REGION Network 21: UNIT 02 FIXTURE 2 PART A PRESENT
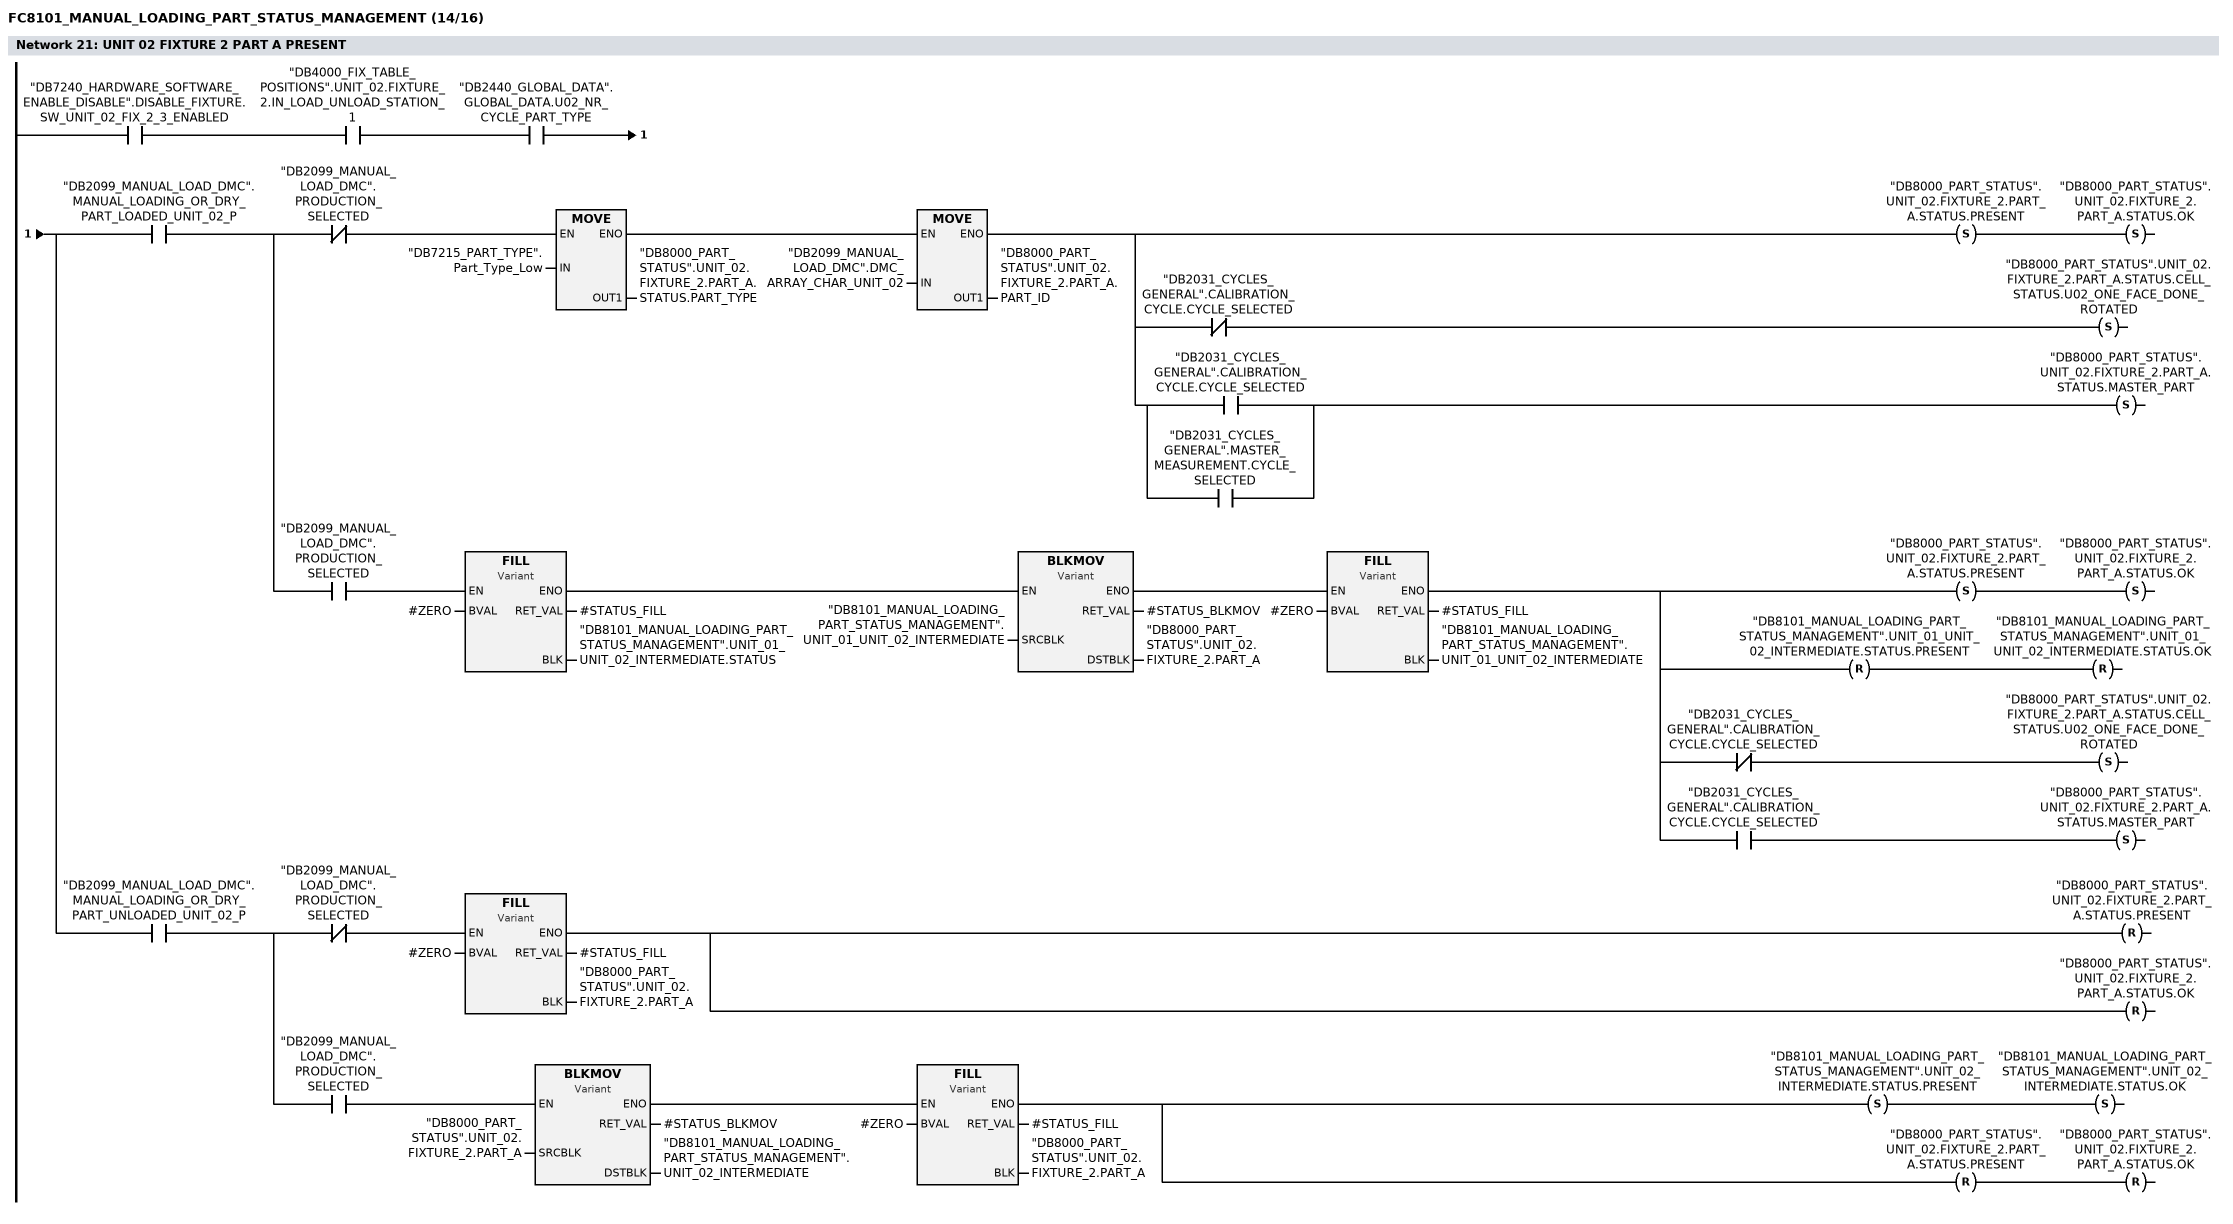
   RUNG wire#powerrail
      Contact( "DB7240_HARDWARE_SOFTWARE_ENABLE_DISABLE".DISABLE_FIXTURE.SW_UNIT_02_FIX_2_3_ENABLED )
      Contact( "DB4000_FIX_TABLE_POSITIONS".UNIT_02.FIXTURE_2.IN_LOAD_UNLOAD_STATION_1 )
      Contact( "DB2440_GLOBAL_DATA".GLOBAL_DATA.U02_NR_CYCLE_PART_TYPE )
      wire#w1
      Contact( "DB2099_MANUAL_LOAD_DMC".MANUAL_LOADING_OR_DRY_PART_LOADED_UNIT_02_P )
      wire#w2
      I_Contact( "DB2099_MANUAL_LOAD_DMC".PRODUCTION_SELECTED )
      { S7_GenerateENO := "TRUE" } Move(in := "DB7215_PART_TYPE".Part_Type_Low, out1 => "DB8000_PART_STATUS".UNIT_02.FIXTURE_2.PART_A.STATUS.PART_TYPE)
      Move(in := "DB2099_MANUAL_LOAD_DMC".DMC_ARRAY_CHAR_UNIT_02, out1 => "DB8000_PART_STATUS".UNIT_02.FIXTURE_2.PART_A.PART_ID)
      wire#w3
      S_Coil( "DB8000_PART_STATUS".UNIT_02.FIXTURE_2.PART_A.STATUS.PRESENT )
      S_Coil( "DB8000_PART_STATUS".UNIT_02.FIXTURE_2.PART_A.STATUS.OK )
   END_RUNG
   RUNG wire#w3
      I_Contact( "DB2031_CYCLES_GENERAL".CALIBRATION_CYCLE.CYCLE_SELECTED )
      S_Coil( "DB8000_PART_STATUS".UNIT_02.FIXTURE_2.PART_A.STATUS.CELL_STATUS.U02_ONE_FACE_DONE_ROTATED )
   END_RUNG
   RUNG wire#w3
      Contact( "DB2031_CYCLES_GENERAL".CALIBRATION_CYCLE.CYCLE_SELECTED )
      wire#w4
      S_Coil( "DB8000_PART_STATUS".UNIT_02.FIXTURE_2.PART_A.STATUS.MASTER_PART )
   END_RUNG
   RUNG wire#w3
      Contact( "DB2031_CYCLES_GENERAL".MASTER_MEASUREMENT.CYCLE_SELECTED )
   END_RUNG wire#w4
   RUNG wire#w2
      Contact( "DB2099_MANUAL_LOAD_DMC".PRODUCTION_SELECTED )
      { S7_Templates := "ptr_type := Variant" } FILL(BVAL := #ZERO, RET_VAL => #STATUS_FILL, BLK => "DB8101_MANUAL_LOADING_PART_STATUS_MANAGEMENT".UNIT_01_UNIT_02_INTERMEDIATE.STATUS)
      { S7_Templates := "blk_type := Variant" } BLKMOV(SRCBLK := "DB8101_MANUAL_LOADING_PART_STATUS_MANAGEMENT".UNIT_01_UNIT_02_INTERMEDIATE, RET_VAL => #STATUS_BLKMOV, DSTBLK => "DB8000_PART_STATUS".UNIT_02.FIXTURE_2.PART_A)
      { S7_Templates := "ptr_type := Variant" } FILL(BVAL := #ZERO, RET_VAL => #STATUS_FILL, BLK => "DB8101_MANUAL_LOADING_PART_STATUS_MANAGEMENT".UNIT_01_UNIT_02_INTERMEDIATE)
      wire#w5
      S_Coil( "DB8000_PART_STATUS".UNIT_02.FIXTURE_2.PART_A.STATUS.PRESENT )
      S_Coil( "DB8000_PART_STATUS".UNIT_02.FIXTURE_2.PART_A.STATUS.OK )
   END_RUNG
   RUNG wire#w5
      R_Coil( "DB8101_MANUAL_LOADING_PART_STATUS_MANAGEMENT".UNIT_01_UNIT_02_INTERMEDIATE.STATUS.PRESENT )
      R_Coil( "DB8101_MANUAL_LOADING_PART_STATUS_MANAGEMENT".UNIT_01_UNIT_02_INTERMEDIATE.STATUS.OK )
   END_RUNG
   RUNG wire#w5
      I_Contact( "DB2031_CYCLES_GENERAL".CALIBRATION_CYCLE.CYCLE_SELECTED )
      S_Coil( "DB8000_PART_STATUS".UNIT_02.FIXTURE_2.PART_A.STATUS.CELL_STATUS.U02_ONE_FACE_DONE_ROTATED )
   END_RUNG
   RUNG wire#w5
      Contact( "DB2031_CYCLES_GENERAL".CALIBRATION_CYCLE.CYCLE_SELECTED )
      S_Coil( "DB8000_PART_STATUS".UNIT_02.FIXTURE_2.PART_A.STATUS.MASTER_PART )
   END_RUNG
   RUNG wire#w1
      Contact( "DB2099_MANUAL_LOAD_DMC".MANUAL_LOADING_OR_DRY_PART_UNLOADED_UNIT_02_P )
      wire#w6
      I_Contact( "DB2099_MANUAL_LOAD_DMC".PRODUCTION_SELECTED )
      { S7_Templates := "ptr_type := Variant" } FILL(BVAL := #ZERO, RET_VAL => #STATUS_FILL, BLK => "DB8000_PART_STATUS".UNIT_02.FIXTURE_2.PART_A)
      wire#w7
      R_Coil( "DB8000_PART_STATUS".UNIT_02.FIXTURE_2.PART_A.STATUS.PRESENT )
   END_RUNG
   RUNG wire#w7
      R_Coil( "DB8000_PART_STATUS".UNIT_02.FIXTURE_2.PART_A.STATUS.OK )
   END_RUNG
   RUNG wire#w6
      Contact( "DB2099_MANUAL_LOAD_DMC".PRODUCTION_SELECTED )
      { S7_Templates := "blk_type := Variant" } BLKMOV(SRCBLK := "DB8000_PART_STATUS".UNIT_02.FIXTURE_2.PART_A, RET_VAL => #STATUS_BLKMOV, DSTBLK => "DB8101_MANUAL_LOADING_PART_STATUS_MANAGEMENT".UNIT_02_INTERMEDIATE)
      { S7_Templates := "ptr_type := Variant" } FILL(BVAL := #ZERO, RET_VAL => #STATUS_FILL, BLK => "DB8000_PART_STATUS".UNIT_02.FIXTURE_2.PART_A)
      wire#w8
      S_Coil( "DB8101_MANUAL_LOADING_PART_STATUS_MANAGEMENT".UNIT_02_INTERMEDIATE.STATUS.PRESENT )
      S_Coil( "DB8101_MANUAL_LOADING_PART_STATUS_MANAGEMENT".UNIT_02_INTERMEDIATE.STATUS.OK )
   END_RUNG
   RUNG wire#w8
      R_Coil( "DB8000_PART_STATUS".UNIT_02.FIXTURE_2.PART_A.STATUS.PRESENT )
      R_Coil( "DB8000_PART_STATUS".UNIT_02.FIXTURE_2.PART_A.STATUS.OK )
   END_RUNG
   // the same network as SCL:
   // ENO of a box is taken as its EN; it also drops when the box reports an error
   #_w1 := "DB7240_HARDWARE_SOFTWARE_ENABLE_DISABLE".DISABLE_FIXTURE.SW_UNIT_02_FIX_2_3_ENABLED AND "DB4000_FIX_TABLE_POSITIONS".UNIT_02.FIXTURE_2.IN_LOAD_UNLOAD_STATION_1 AND "DB2440_GLOBAL_DATA".GLOBAL_DATA.U02_NR_CYCLE_PART_TYPE;
   #_w2 := #_w1 AND "DB2099_MANUAL_LOAD_DMC".MANUAL_LOADING_OR_DRY_PART_LOADED_UNIT_02_P;
   #_w3 := #_w2 AND NOT "DB2099_MANUAL_LOAD_DMC".PRODUCTION_SELECTED;
   IF #_w3 THEN
       "DB8000_PART_STATUS".UNIT_02.FIXTURE_2.PART_A.STATUS.PART_TYPE := "DB7215_PART_TYPE".Part_Type_Low;
       "DB8000_PART_STATUS".UNIT_02.FIXTURE_2.PART_A.PART_ID := "DB2099_MANUAL_LOAD_DMC".DMC_ARRAY_CHAR_UNIT_02;
       "DB8000_PART_STATUS".UNIT_02.FIXTURE_2.PART_A.STATUS.PRESENT := TRUE;
       "DB8000_PART_STATUS".UNIT_02.FIXTURE_2.PART_A.STATUS.OK := TRUE;
   END_IF;
   IF #_w3 AND NOT "DB2031_CYCLES_GENERAL".CALIBRATION_CYCLE.CYCLE_SELECTED THEN
       "DB8000_PART_STATUS".UNIT_02.FIXTURE_2.PART_A.STATUS.CELL_STATUS.U02_ONE_FACE_DONE_ROTATED := TRUE;
   END_IF;
   IF #_w3 AND ("DB2031_CYCLES_GENERAL".CALIBRATION_CYCLE.CYCLE_SELECTED OR "DB2031_CYCLES_GENERAL".MASTER_MEASUREMENT.CYCLE_SELECTED) THEN
       "DB8000_PART_STATUS".UNIT_02.FIXTURE_2.PART_A.STATUS.MASTER_PART := TRUE;
   END_IF;
   #_w4 := #_w2 AND "DB2099_MANUAL_LOAD_DMC".PRODUCTION_SELECTED;
   #STATUS_FILL := FILL(EN := #_w4,
                        BVAL := #ZERO,
                        BLK => "DB8101_MANUAL_LOADING_PART_STATUS_MANAGEMENT".UNIT_01_UNIT_02_INTERMEDIATE.STATUS,
                        ENO => #_w5);
   #STATUS_BLKMOV := BLKMOV(EN := #_w5,
                           SRCBLK := "DB8101_MANUAL_LOADING_PART_STATUS_MANAGEMENT".UNIT_01_UNIT_02_INTERMEDIATE,
                           DSTBLK => "DB8000_PART_STATUS".UNIT_02.FIXTURE_2.PART_A,
                           ENO => #_w6);
   #STATUS_FILL := FILL(EN := #_w6,
                        BVAL := #ZERO,
                        BLK => "DB8101_MANUAL_LOADING_PART_STATUS_MANAGEMENT".UNIT_01_UNIT_02_INTERMEDIATE,
                        ENO => #_w7);
   IF #_w7 THEN
       "DB8000_PART_STATUS".UNIT_02.FIXTURE_2.PART_A.STATUS.PRESENT := TRUE;
       "DB8000_PART_STATUS".UNIT_02.FIXTURE_2.PART_A.STATUS.OK := TRUE;
       "DB8101_MANUAL_LOADING_PART_STATUS_MANAGEMENT".UNIT_01_UNIT_02_INTERMEDIATE.STATUS.PRESENT := FALSE;
       "DB8101_MANUAL_LOADING_PART_STATUS_MANAGEMENT".UNIT_01_UNIT_02_INTERMEDIATE.STATUS.OK := FALSE;
   END_IF;
   IF #_w7 AND NOT "DB2031_CYCLES_GENERAL".CALIBRATION_CYCLE.CYCLE_SELECTED THEN
       "DB8000_PART_STATUS".UNIT_02.FIXTURE_2.PART_A.STATUS.CELL_STATUS.U02_ONE_FACE_DONE_ROTATED := TRUE;
   END_IF;
   IF #_w7 AND "DB2031_CYCLES_GENERAL".CALIBRATION_CYCLE.CYCLE_SELECTED THEN
       "DB8000_PART_STATUS".UNIT_02.FIXTURE_2.PART_A.STATUS.MASTER_PART := TRUE;
   END_IF;
   #_w8 := #_w1 AND "DB2099_MANUAL_LOAD_DMC".MANUAL_LOADING_OR_DRY_PART_UNLOADED_UNIT_02_P;
   #STATUS_FILL := FILL(EN := #_w8 AND NOT "DB2099_MANUAL_LOAD_DMC".PRODUCTION_SELECTED,
                        BVAL := #ZERO,
                        BLK => "DB8000_PART_STATUS".UNIT_02.FIXTURE_2.PART_A,
                        ENO => #_w9);
   IF #_w9 THEN
       "DB8000_PART_STATUS".UNIT_02.FIXTURE_2.PART_A.STATUS.PRESENT := FALSE;
       "DB8000_PART_STATUS".UNIT_02.FIXTURE_2.PART_A.STATUS.OK := FALSE;
   END_IF;
   #STATUS_BLKMOV := BLKMOV(EN := #_w8 AND "DB2099_MANUAL_LOAD_DMC".PRODUCTION_SELECTED,
                           SRCBLK := "DB8000_PART_STATUS".UNIT_02.FIXTURE_2.PART_A,
                           DSTBLK => "DB8101_MANUAL_LOADING_PART_STATUS_MANAGEMENT".UNIT_02_INTERMEDIATE,
                           ENO => #_w10);
   #STATUS_FILL := FILL(EN := #_w10,
                        BVAL := #ZERO,
                        BLK => "DB8000_PART_STATUS".UNIT_02.FIXTURE_2.PART_A,
                        ENO => #_w11);
   IF #_w11 THEN
       "DB8101_MANUAL_LOADING_PART_STATUS_MANAGEMENT".UNIT_02_INTERMEDIATE.STATUS.PRESENT := TRUE;
       "DB8101_MANUAL_LOADING_PART_STATUS_MANAGEMENT".UNIT_02_INTERMEDIATE.STATUS.OK := TRUE;
       "DB8000_PART_STATUS".UNIT_02.FIXTURE_2.PART_A.STATUS.PRESENT := FALSE;
       "DB8000_PART_STATUS".UNIT_02.FIXTURE_2.PART_A.STATUS.OK := FALSE;
   END_IF;
END_REGION

REGION Network 22: UNIT 02 FIXTURE 3 PART A PRESENT
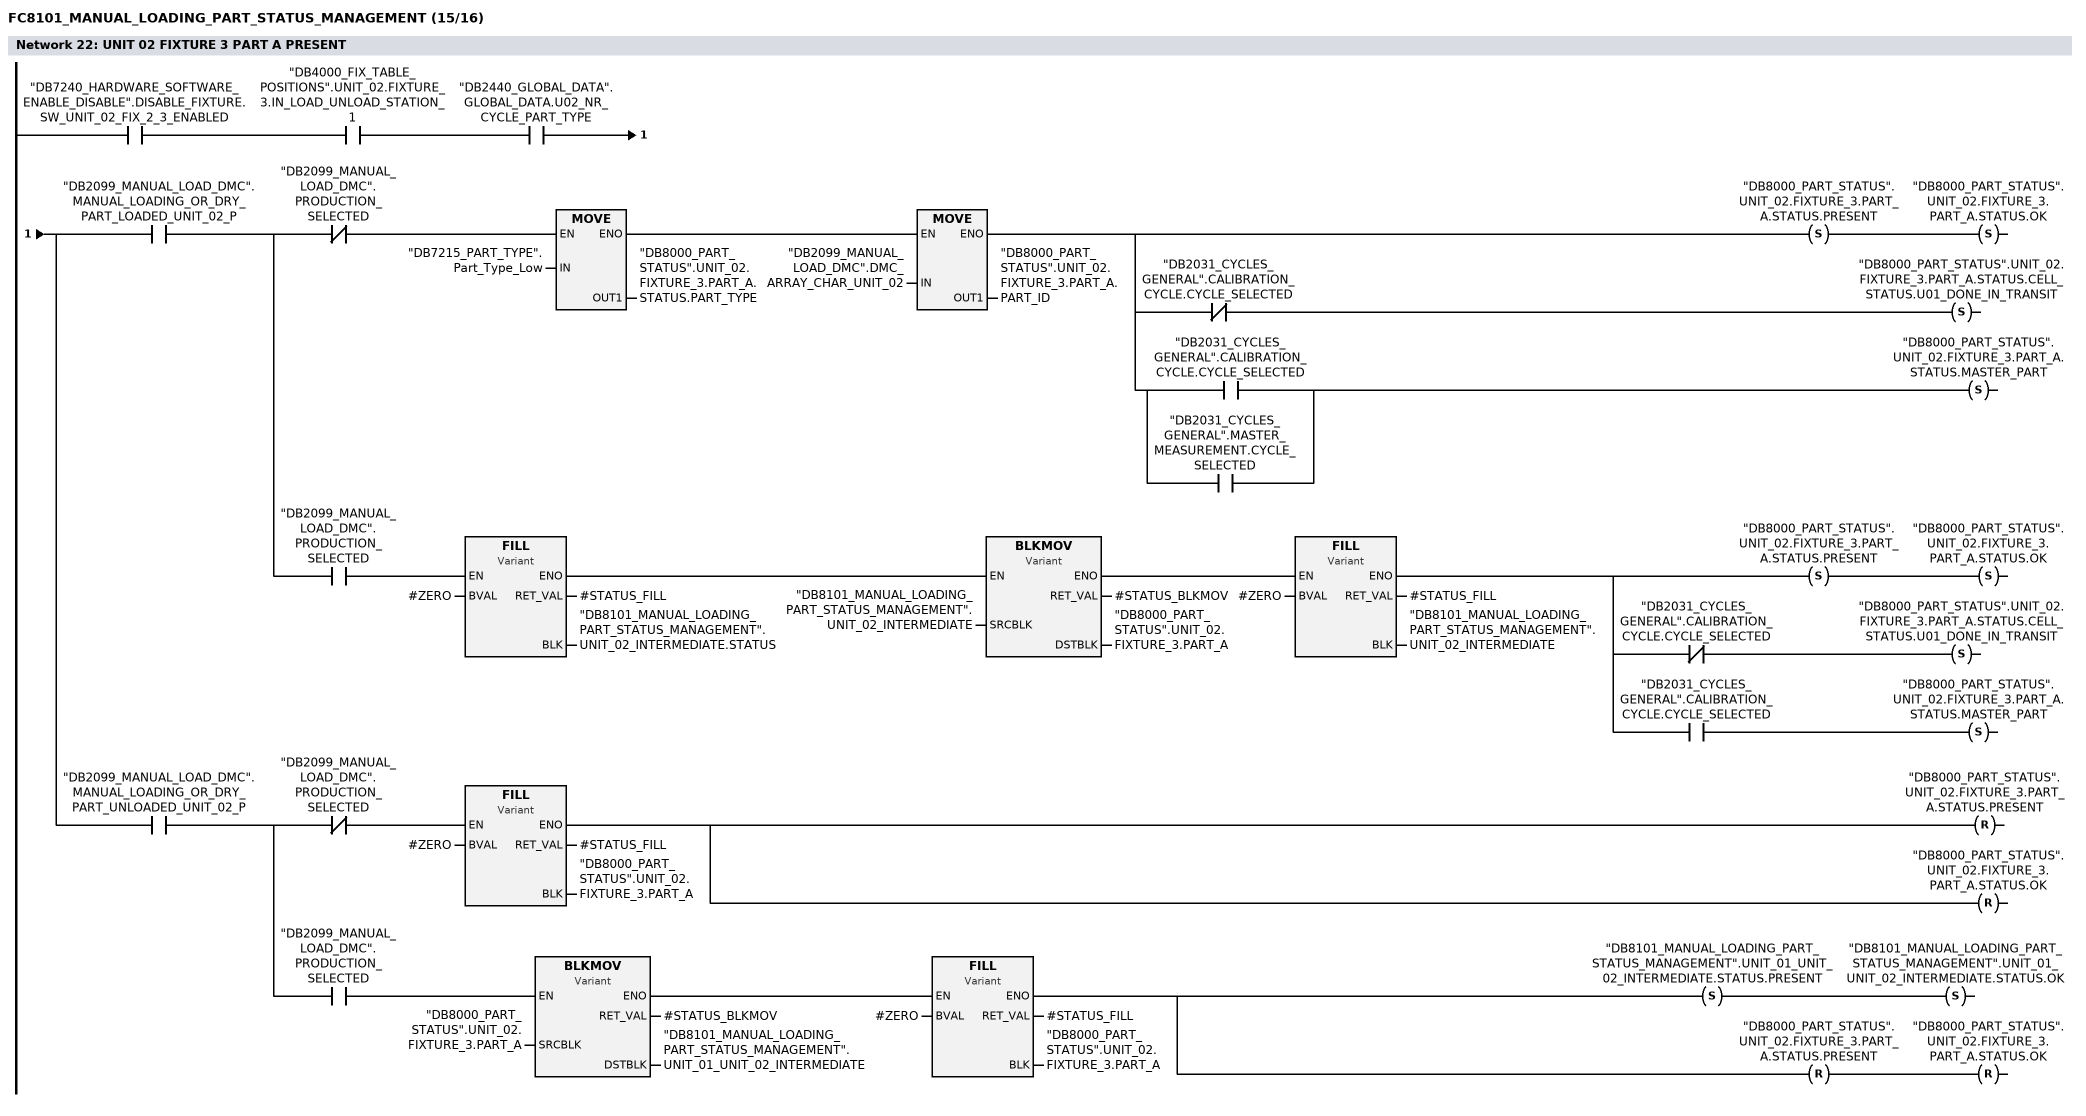
   RUNG wire#powerrail
      Contact( "DB7240_HARDWARE_SOFTWARE_ENABLE_DISABLE".DISABLE_FIXTURE.SW_UNIT_02_FIX_2_3_ENABLED )
      Contact( "DB4000_FIX_TABLE_POSITIONS".UNIT_02.FIXTURE_3.IN_LOAD_UNLOAD_STATION_1 )
      Contact( "DB2440_GLOBAL_DATA".GLOBAL_DATA.U02_NR_CYCLE_PART_TYPE )
      wire#w1
      Contact( "DB2099_MANUAL_LOAD_DMC".MANUAL_LOADING_OR_DRY_PART_LOADED_UNIT_02_P )
      wire#w2
      I_Contact( "DB2099_MANUAL_LOAD_DMC".PRODUCTION_SELECTED )
      { S7_GenerateENO := "TRUE" } Move(in := "DB7215_PART_TYPE".Part_Type_Low, out1 => "DB8000_PART_STATUS".UNIT_02.FIXTURE_3.PART_A.STATUS.PART_TYPE)
      Move(in := "DB2099_MANUAL_LOAD_DMC".DMC_ARRAY_CHAR_UNIT_02, out1 => "DB8000_PART_STATUS".UNIT_02.FIXTURE_3.PART_A.PART_ID)
      wire#w3
      S_Coil( "DB8000_PART_STATUS".UNIT_02.FIXTURE_3.PART_A.STATUS.PRESENT )
      S_Coil( "DB8000_PART_STATUS".UNIT_02.FIXTURE_3.PART_A.STATUS.OK )
   END_RUNG
   RUNG wire#w3
      I_Contact( "DB2031_CYCLES_GENERAL".CALIBRATION_CYCLE.CYCLE_SELECTED )
      S_Coil( "DB8000_PART_STATUS".UNIT_02.FIXTURE_3.PART_A.STATUS.CELL_STATUS.U01_DONE_IN_TRANSIT )
   END_RUNG
   RUNG wire#w3
      Contact( "DB2031_CYCLES_GENERAL".CALIBRATION_CYCLE.CYCLE_SELECTED )
      wire#w4
      S_Coil( "DB8000_PART_STATUS".UNIT_02.FIXTURE_3.PART_A.STATUS.MASTER_PART )
   END_RUNG
   RUNG wire#w3
      Contact( "DB2031_CYCLES_GENERAL".MASTER_MEASUREMENT.CYCLE_SELECTED )
   END_RUNG wire#w4
   RUNG wire#w2
      Contact( "DB2099_MANUAL_LOAD_DMC".PRODUCTION_SELECTED )
      { S7_Templates := "ptr_type := Variant" } FILL(BVAL := #ZERO, RET_VAL => #STATUS_FILL, BLK => "DB8101_MANUAL_LOADING_PART_STATUS_MANAGEMENT".UNIT_02_INTERMEDIATE.STATUS)
      { S7_Templates := "blk_type := Variant" } BLKMOV(SRCBLK := "DB8101_MANUAL_LOADING_PART_STATUS_MANAGEMENT".UNIT_02_INTERMEDIATE, RET_VAL => #STATUS_BLKMOV, DSTBLK => "DB8000_PART_STATUS".UNIT_02.FIXTURE_3.PART_A)
      { S7_Templates := "ptr_type := Variant" } FILL(BVAL := #ZERO, RET_VAL => #STATUS_FILL, BLK => "DB8101_MANUAL_LOADING_PART_STATUS_MANAGEMENT".UNIT_02_INTERMEDIATE)
      wire#w5
      S_Coil( "DB8000_PART_STATUS".UNIT_02.FIXTURE_3.PART_A.STATUS.PRESENT )
      S_Coil( "DB8000_PART_STATUS".UNIT_02.FIXTURE_3.PART_A.STATUS.OK )
   END_RUNG
   RUNG wire#w5
      I_Contact( "DB2031_CYCLES_GENERAL".CALIBRATION_CYCLE.CYCLE_SELECTED )
      S_Coil( "DB8000_PART_STATUS".UNIT_02.FIXTURE_3.PART_A.STATUS.CELL_STATUS.U01_DONE_IN_TRANSIT )
   END_RUNG
   RUNG wire#w5
      Contact( "DB2031_CYCLES_GENERAL".CALIBRATION_CYCLE.CYCLE_SELECTED )
      S_Coil( "DB8000_PART_STATUS".UNIT_02.FIXTURE_3.PART_A.STATUS.MASTER_PART )
   END_RUNG
   RUNG wire#w1
      Contact( "DB2099_MANUAL_LOAD_DMC".MANUAL_LOADING_OR_DRY_PART_UNLOADED_UNIT_02_P )
      wire#w6
      I_Contact( "DB2099_MANUAL_LOAD_DMC".PRODUCTION_SELECTED )
      { S7_Templates := "ptr_type := Variant" } FILL(BVAL := #ZERO, RET_VAL => #STATUS_FILL, BLK => "DB8000_PART_STATUS".UNIT_02.FIXTURE_3.PART_A)
      wire#w7
      R_Coil( "DB8000_PART_STATUS".UNIT_02.FIXTURE_3.PART_A.STATUS.PRESENT )
   END_RUNG
   RUNG wire#w7
      R_Coil( "DB8000_PART_STATUS".UNIT_02.FIXTURE_3.PART_A.STATUS.OK )
   END_RUNG
   RUNG wire#w6
      Contact( "DB2099_MANUAL_LOAD_DMC".PRODUCTION_SELECTED )
      { S7_Templates := "blk_type := Variant" } BLKMOV(SRCBLK := "DB8000_PART_STATUS".UNIT_02.FIXTURE_3.PART_A, RET_VAL => #STATUS_BLKMOV, DSTBLK => "DB8101_MANUAL_LOADING_PART_STATUS_MANAGEMENT".UNIT_01_UNIT_02_INTERMEDIATE)
      { S7_Templates := "ptr_type := Variant" } FILL(BVAL := #ZERO, RET_VAL => #STATUS_FILL, BLK => "DB8000_PART_STATUS".UNIT_02.FIXTURE_3.PART_A)
      wire#w8
      S_Coil( "DB8101_MANUAL_LOADING_PART_STATUS_MANAGEMENT".UNIT_01_UNIT_02_INTERMEDIATE.STATUS.PRESENT )
      S_Coil( "DB8101_MANUAL_LOADING_PART_STATUS_MANAGEMENT".UNIT_01_UNIT_02_INTERMEDIATE.STATUS.OK )
   END_RUNG
   RUNG wire#w8
      R_Coil( "DB8000_PART_STATUS".UNIT_02.FIXTURE_3.PART_A.STATUS.PRESENT )
      R_Coil( "DB8000_PART_STATUS".UNIT_02.FIXTURE_3.PART_A.STATUS.OK )
   END_RUNG
   // the same network as SCL:
   // ENO of a box is taken as its EN; it also drops when the box reports an error
   #_w1 := "DB7240_HARDWARE_SOFTWARE_ENABLE_DISABLE".DISABLE_FIXTURE.SW_UNIT_02_FIX_2_3_ENABLED AND "DB4000_FIX_TABLE_POSITIONS".UNIT_02.FIXTURE_3.IN_LOAD_UNLOAD_STATION_1 AND "DB2440_GLOBAL_DATA".GLOBAL_DATA.U02_NR_CYCLE_PART_TYPE;
   #_w2 := #_w1 AND "DB2099_MANUAL_LOAD_DMC".MANUAL_LOADING_OR_DRY_PART_LOADED_UNIT_02_P;
   #_w3 := #_w2 AND NOT "DB2099_MANUAL_LOAD_DMC".PRODUCTION_SELECTED;
   IF #_w3 THEN
       "DB8000_PART_STATUS".UNIT_02.FIXTURE_3.PART_A.STATUS.PART_TYPE := "DB7215_PART_TYPE".Part_Type_Low;
       "DB8000_PART_STATUS".UNIT_02.FIXTURE_3.PART_A.PART_ID := "DB2099_MANUAL_LOAD_DMC".DMC_ARRAY_CHAR_UNIT_02;
       "DB8000_PART_STATUS".UNIT_02.FIXTURE_3.PART_A.STATUS.PRESENT := TRUE;
       "DB8000_PART_STATUS".UNIT_02.FIXTURE_3.PART_A.STATUS.OK := TRUE;
   END_IF;
   IF #_w3 AND NOT "DB2031_CYCLES_GENERAL".CALIBRATION_CYCLE.CYCLE_SELECTED THEN
       "DB8000_PART_STATUS".UNIT_02.FIXTURE_3.PART_A.STATUS.CELL_STATUS.U01_DONE_IN_TRANSIT := TRUE;
   END_IF;
   IF #_w3 AND ("DB2031_CYCLES_GENERAL".CALIBRATION_CYCLE.CYCLE_SELECTED OR "DB2031_CYCLES_GENERAL".MASTER_MEASUREMENT.CYCLE_SELECTED) THEN
       "DB8000_PART_STATUS".UNIT_02.FIXTURE_3.PART_A.STATUS.MASTER_PART := TRUE;
   END_IF;
   #_w4 := #_w2 AND "DB2099_MANUAL_LOAD_DMC".PRODUCTION_SELECTED;
   #STATUS_FILL := FILL(EN := #_w4,
                        BVAL := #ZERO,
                        BLK => "DB8101_MANUAL_LOADING_PART_STATUS_MANAGEMENT".UNIT_02_INTERMEDIATE.STATUS,
                        ENO => #_w5);
   #STATUS_BLKMOV := BLKMOV(EN := #_w5,
                           SRCBLK := "DB8101_MANUAL_LOADING_PART_STATUS_MANAGEMENT".UNIT_02_INTERMEDIATE,
                           DSTBLK => "DB8000_PART_STATUS".UNIT_02.FIXTURE_3.PART_A,
                           ENO => #_w6);
   #STATUS_FILL := FILL(EN := #_w6,
                        BVAL := #ZERO,
                        BLK => "DB8101_MANUAL_LOADING_PART_STATUS_MANAGEMENT".UNIT_02_INTERMEDIATE,
                        ENO => #_w7);
   IF #_w7 THEN
       "DB8000_PART_STATUS".UNIT_02.FIXTURE_3.PART_A.STATUS.PRESENT := TRUE;
       "DB8000_PART_STATUS".UNIT_02.FIXTURE_3.PART_A.STATUS.OK := TRUE;
   END_IF;
   IF #_w7 AND NOT "DB2031_CYCLES_GENERAL".CALIBRATION_CYCLE.CYCLE_SELECTED THEN
       "DB8000_PART_STATUS".UNIT_02.FIXTURE_3.PART_A.STATUS.CELL_STATUS.U01_DONE_IN_TRANSIT := TRUE;
   END_IF;
   IF #_w7 AND "DB2031_CYCLES_GENERAL".CALIBRATION_CYCLE.CYCLE_SELECTED THEN
       "DB8000_PART_STATUS".UNIT_02.FIXTURE_3.PART_A.STATUS.MASTER_PART := TRUE;
   END_IF;
   #_w8 := #_w1 AND "DB2099_MANUAL_LOAD_DMC".MANUAL_LOADING_OR_DRY_PART_UNLOADED_UNIT_02_P;
   #STATUS_FILL := FILL(EN := #_w8 AND NOT "DB2099_MANUAL_LOAD_DMC".PRODUCTION_SELECTED,
                        BVAL := #ZERO,
                        BLK => "DB8000_PART_STATUS".UNIT_02.FIXTURE_3.PART_A,
                        ENO => #_w9);
   IF #_w9 THEN
       "DB8000_PART_STATUS".UNIT_02.FIXTURE_3.PART_A.STATUS.PRESENT := FALSE;
       "DB8000_PART_STATUS".UNIT_02.FIXTURE_3.PART_A.STATUS.OK := FALSE;
   END_IF;
   #STATUS_BLKMOV := BLKMOV(EN := #_w8 AND "DB2099_MANUAL_LOAD_DMC".PRODUCTION_SELECTED,
                           SRCBLK := "DB8000_PART_STATUS".UNIT_02.FIXTURE_3.PART_A,
                           DSTBLK => "DB8101_MANUAL_LOADING_PART_STATUS_MANAGEMENT".UNIT_01_UNIT_02_INTERMEDIATE,
                           ENO => #_w10);
   #STATUS_FILL := FILL(EN := #_w10,
                        BVAL := #ZERO,
                        BLK => "DB8000_PART_STATUS".UNIT_02.FIXTURE_3.PART_A,
                        ENO => #_w11);
   IF #_w11 THEN
       "DB8101_MANUAL_LOADING_PART_STATUS_MANAGEMENT".UNIT_01_UNIT_02_INTERMEDIATE.STATUS.PRESENT := TRUE;
       "DB8101_MANUAL_LOADING_PART_STATUS_MANAGEMENT".UNIT_01_UNIT_02_INTERMEDIATE.STATUS.OK := TRUE;
       "DB8000_PART_STATUS".UNIT_02.FIXTURE_3.PART_A.STATUS.PRESENT := FALSE;
       "DB8000_PART_STATUS".UNIT_02.FIXTURE_3.PART_A.STATUS.OK := FALSE;
   END_IF;
END_REGION

REGION Network 23: UNIT 02 FIXTURE 4 PART A PRESENT
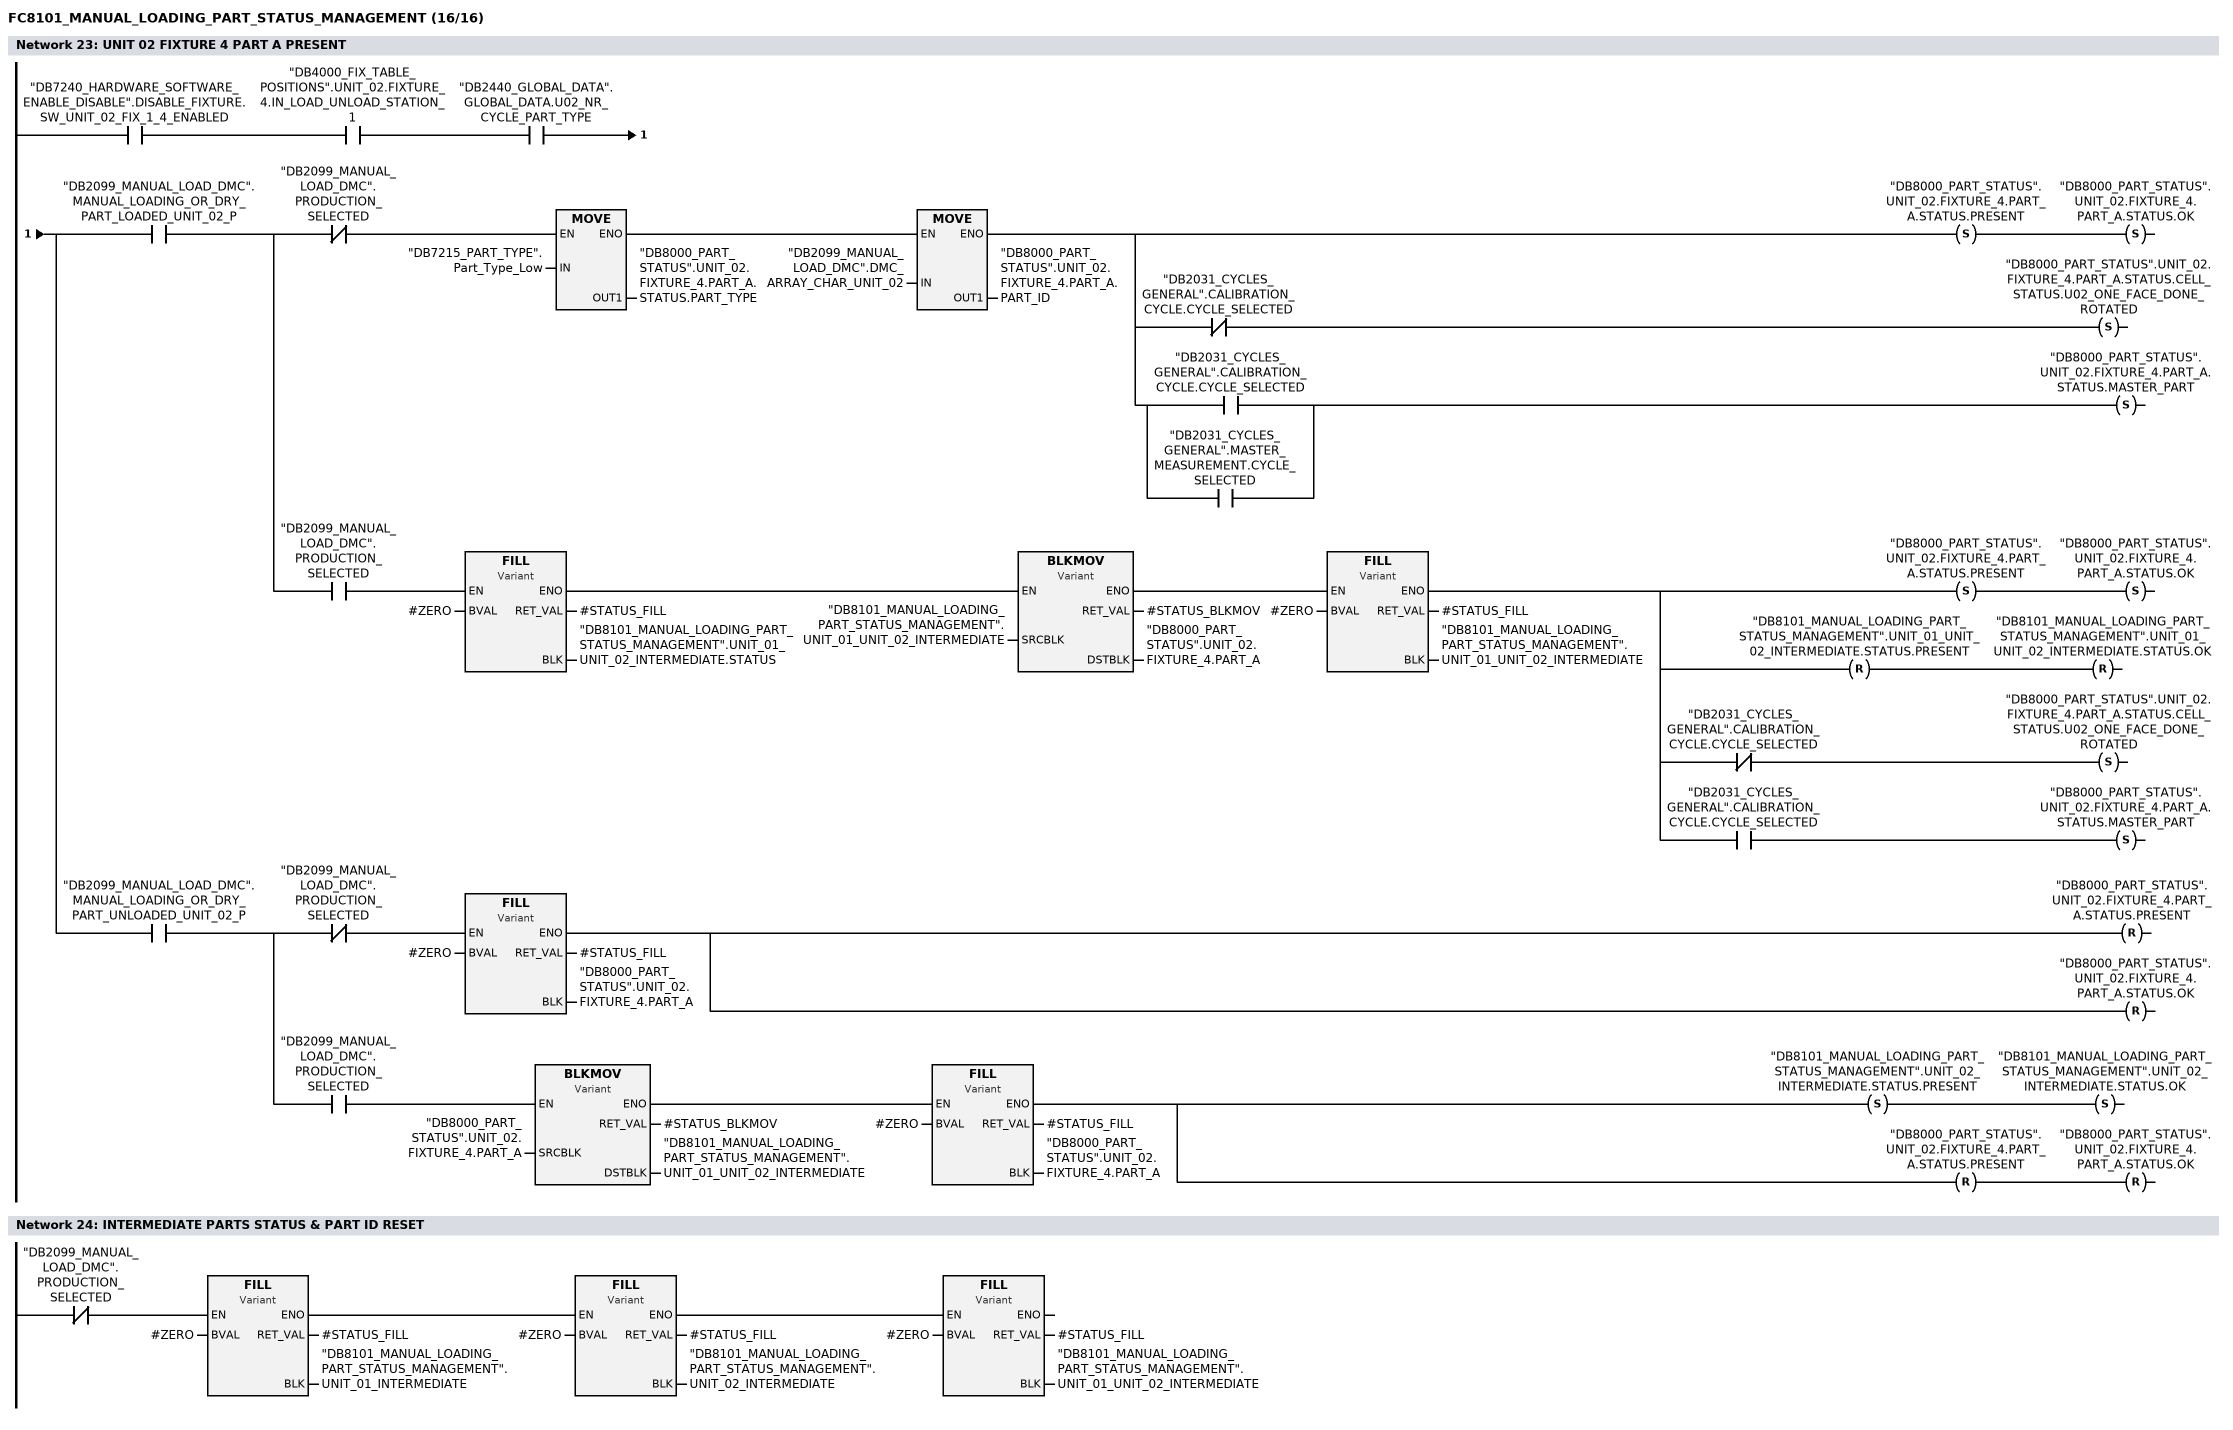
   RUNG wire#powerrail
      Contact( "DB7240_HARDWARE_SOFTWARE_ENABLE_DISABLE".DISABLE_FIXTURE.SW_UNIT_02_FIX_1_4_ENABLED )
      Contact( "DB4000_FIX_TABLE_POSITIONS".UNIT_02.FIXTURE_4.IN_LOAD_UNLOAD_STATION_1 )
      Contact( "DB2440_GLOBAL_DATA".GLOBAL_DATA.U02_NR_CYCLE_PART_TYPE )
      wire#w1
      Contact( "DB2099_MANUAL_LOAD_DMC".MANUAL_LOADING_OR_DRY_PART_LOADED_UNIT_02_P )
      wire#w2
      I_Contact( "DB2099_MANUAL_LOAD_DMC".PRODUCTION_SELECTED )
      { S7_GenerateENO := "TRUE" } Move(in := "DB7215_PART_TYPE".Part_Type_Low, out1 => "DB8000_PART_STATUS".UNIT_02.FIXTURE_4.PART_A.STATUS.PART_TYPE)
      Move(in := "DB2099_MANUAL_LOAD_DMC".DMC_ARRAY_CHAR_UNIT_02, out1 => "DB8000_PART_STATUS".UNIT_02.FIXTURE_4.PART_A.PART_ID)
      wire#w3
      S_Coil( "DB8000_PART_STATUS".UNIT_02.FIXTURE_4.PART_A.STATUS.PRESENT )
      S_Coil( "DB8000_PART_STATUS".UNIT_02.FIXTURE_4.PART_A.STATUS.OK )
   END_RUNG
   RUNG wire#w3
      I_Contact( "DB2031_CYCLES_GENERAL".CALIBRATION_CYCLE.CYCLE_SELECTED )
      S_Coil( "DB8000_PART_STATUS".UNIT_02.FIXTURE_4.PART_A.STATUS.CELL_STATUS.U02_ONE_FACE_DONE_ROTATED )
   END_RUNG
   RUNG wire#w3
      Contact( "DB2031_CYCLES_GENERAL".CALIBRATION_CYCLE.CYCLE_SELECTED )
      wire#w4
      S_Coil( "DB8000_PART_STATUS".UNIT_02.FIXTURE_4.PART_A.STATUS.MASTER_PART )
   END_RUNG
   RUNG wire#w3
      Contact( "DB2031_CYCLES_GENERAL".MASTER_MEASUREMENT.CYCLE_SELECTED )
   END_RUNG wire#w4
   RUNG wire#w2
      Contact( "DB2099_MANUAL_LOAD_DMC".PRODUCTION_SELECTED )
      { S7_Templates := "ptr_type := Variant" } FILL(BVAL := #ZERO, RET_VAL => #STATUS_FILL, BLK => "DB8101_MANUAL_LOADING_PART_STATUS_MANAGEMENT".UNIT_01_UNIT_02_INTERMEDIATE.STATUS)
      { S7_Templates := "blk_type := Variant" } BLKMOV(SRCBLK := "DB8101_MANUAL_LOADING_PART_STATUS_MANAGEMENT".UNIT_01_UNIT_02_INTERMEDIATE, RET_VAL => #STATUS_BLKMOV, DSTBLK => "DB8000_PART_STATUS".UNIT_02.FIXTURE_4.PART_A)
      { S7_Templates := "ptr_type := Variant" } FILL(BVAL := #ZERO, RET_VAL => #STATUS_FILL, BLK => "DB8101_MANUAL_LOADING_PART_STATUS_MANAGEMENT".UNIT_01_UNIT_02_INTERMEDIATE)
      wire#w5
      S_Coil( "DB8000_PART_STATUS".UNIT_02.FIXTURE_4.PART_A.STATUS.PRESENT )
      S_Coil( "DB8000_PART_STATUS".UNIT_02.FIXTURE_4.PART_A.STATUS.OK )
   END_RUNG
   RUNG wire#w5
      R_Coil( "DB8101_MANUAL_LOADING_PART_STATUS_MANAGEMENT".UNIT_01_UNIT_02_INTERMEDIATE.STATUS.PRESENT )
      R_Coil( "DB8101_MANUAL_LOADING_PART_STATUS_MANAGEMENT".UNIT_01_UNIT_02_INTERMEDIATE.STATUS.OK )
   END_RUNG
   RUNG wire#w5
      I_Contact( "DB2031_CYCLES_GENERAL".CALIBRATION_CYCLE.CYCLE_SELECTED )
      S_Coil( "DB8000_PART_STATUS".UNIT_02.FIXTURE_4.PART_A.STATUS.CELL_STATUS.U02_ONE_FACE_DONE_ROTATED )
   END_RUNG
   RUNG wire#w5
      Contact( "DB2031_CYCLES_GENERAL".CALIBRATION_CYCLE.CYCLE_SELECTED )
      S_Coil( "DB8000_PART_STATUS".UNIT_02.FIXTURE_4.PART_A.STATUS.MASTER_PART )
   END_RUNG
   RUNG wire#w1
      Contact( "DB2099_MANUAL_LOAD_DMC".MANUAL_LOADING_OR_DRY_PART_UNLOADED_UNIT_02_P )
      wire#w6
      I_Contact( "DB2099_MANUAL_LOAD_DMC".PRODUCTION_SELECTED )
      { S7_Templates := "ptr_type := Variant" } FILL(BVAL := #ZERO, RET_VAL => #STATUS_FILL, BLK => "DB8000_PART_STATUS".UNIT_02.FIXTURE_4.PART_A)
      wire#w7
      R_Coil( "DB8000_PART_STATUS".UNIT_02.FIXTURE_4.PART_A.STATUS.PRESENT )
   END_RUNG
   RUNG wire#w7
      R_Coil( "DB8000_PART_STATUS".UNIT_02.FIXTURE_4.PART_A.STATUS.OK )
   END_RUNG
   RUNG wire#w6
      Contact( "DB2099_MANUAL_LOAD_DMC".PRODUCTION_SELECTED )
      { S7_Templates := "blk_type := Variant" } BLKMOV(SRCBLK := "DB8000_PART_STATUS".UNIT_02.FIXTURE_4.PART_A, RET_VAL => #STATUS_BLKMOV, DSTBLK => "DB8101_MANUAL_LOADING_PART_STATUS_MANAGEMENT".UNIT_01_UNIT_02_INTERMEDIATE)
      { S7_Templates := "ptr_type := Variant" } FILL(BVAL := #ZERO, RET_VAL => #STATUS_FILL, BLK => "DB8000_PART_STATUS".UNIT_02.FIXTURE_4.PART_A)
      wire#w8
      S_Coil( "DB8101_MANUAL_LOADING_PART_STATUS_MANAGEMENT".UNIT_02_INTERMEDIATE.STATUS.PRESENT )
      S_Coil( "DB8101_MANUAL_LOADING_PART_STATUS_MANAGEMENT".UNIT_02_INTERMEDIATE.STATUS.OK )
   END_RUNG
   RUNG wire#w8
      R_Coil( "DB8000_PART_STATUS".UNIT_02.FIXTURE_4.PART_A.STATUS.PRESENT )
      R_Coil( "DB8000_PART_STATUS".UNIT_02.FIXTURE_4.PART_A.STATUS.OK )
   END_RUNG
   // the same network as SCL:
   // ENO of a box is taken as its EN; it also drops when the box reports an error
   #_w1 := "DB7240_HARDWARE_SOFTWARE_ENABLE_DISABLE".DISABLE_FIXTURE.SW_UNIT_02_FIX_1_4_ENABLED AND "DB4000_FIX_TABLE_POSITIONS".UNIT_02.FIXTURE_4.IN_LOAD_UNLOAD_STATION_1 AND "DB2440_GLOBAL_DATA".GLOBAL_DATA.U02_NR_CYCLE_PART_TYPE;
   #_w2 := #_w1 AND "DB2099_MANUAL_LOAD_DMC".MANUAL_LOADING_OR_DRY_PART_LOADED_UNIT_02_P;
   #_w3 := #_w2 AND NOT "DB2099_MANUAL_LOAD_DMC".PRODUCTION_SELECTED;
   IF #_w3 THEN
       "DB8000_PART_STATUS".UNIT_02.FIXTURE_4.PART_A.STATUS.PART_TYPE := "DB7215_PART_TYPE".Part_Type_Low;
       "DB8000_PART_STATUS".UNIT_02.FIXTURE_4.PART_A.PART_ID := "DB2099_MANUAL_LOAD_DMC".DMC_ARRAY_CHAR_UNIT_02;
       "DB8000_PART_STATUS".UNIT_02.FIXTURE_4.PART_A.STATUS.PRESENT := TRUE;
       "DB8000_PART_STATUS".UNIT_02.FIXTURE_4.PART_A.STATUS.OK := TRUE;
   END_IF;
   IF #_w3 AND NOT "DB2031_CYCLES_GENERAL".CALIBRATION_CYCLE.CYCLE_SELECTED THEN
       "DB8000_PART_STATUS".UNIT_02.FIXTURE_4.PART_A.STATUS.CELL_STATUS.U02_ONE_FACE_DONE_ROTATED := TRUE;
   END_IF;
   IF #_w3 AND ("DB2031_CYCLES_GENERAL".CALIBRATION_CYCLE.CYCLE_SELECTED OR "DB2031_CYCLES_GENERAL".MASTER_MEASUREMENT.CYCLE_SELECTED) THEN
       "DB8000_PART_STATUS".UNIT_02.FIXTURE_4.PART_A.STATUS.MASTER_PART := TRUE;
   END_IF;
   #_w4 := #_w2 AND "DB2099_MANUAL_LOAD_DMC".PRODUCTION_SELECTED;
   #STATUS_FILL := FILL(EN := #_w4,
                        BVAL := #ZERO,
                        BLK => "DB8101_MANUAL_LOADING_PART_STATUS_MANAGEMENT".UNIT_01_UNIT_02_INTERMEDIATE.STATUS,
                        ENO => #_w5);
   #STATUS_BLKMOV := BLKMOV(EN := #_w5,
                           SRCBLK := "DB8101_MANUAL_LOADING_PART_STATUS_MANAGEMENT".UNIT_01_UNIT_02_INTERMEDIATE,
                           DSTBLK => "DB8000_PART_STATUS".UNIT_02.FIXTURE_4.PART_A,
                           ENO => #_w6);
   #STATUS_FILL := FILL(EN := #_w6,
                        BVAL := #ZERO,
                        BLK => "DB8101_MANUAL_LOADING_PART_STATUS_MANAGEMENT".UNIT_01_UNIT_02_INTERMEDIATE,
                        ENO => #_w7);
   IF #_w7 THEN
       "DB8000_PART_STATUS".UNIT_02.FIXTURE_4.PART_A.STATUS.PRESENT := TRUE;
       "DB8000_PART_STATUS".UNIT_02.FIXTURE_4.PART_A.STATUS.OK := TRUE;
       "DB8101_MANUAL_LOADING_PART_STATUS_MANAGEMENT".UNIT_01_UNIT_02_INTERMEDIATE.STATUS.PRESENT := FALSE;
       "DB8101_MANUAL_LOADING_PART_STATUS_MANAGEMENT".UNIT_01_UNIT_02_INTERMEDIATE.STATUS.OK := FALSE;
   END_IF;
   IF #_w7 AND NOT "DB2031_CYCLES_GENERAL".CALIBRATION_CYCLE.CYCLE_SELECTED THEN
       "DB8000_PART_STATUS".UNIT_02.FIXTURE_4.PART_A.STATUS.CELL_STATUS.U02_ONE_FACE_DONE_ROTATED := TRUE;
   END_IF;
   IF #_w7 AND "DB2031_CYCLES_GENERAL".CALIBRATION_CYCLE.CYCLE_SELECTED THEN
       "DB8000_PART_STATUS".UNIT_02.FIXTURE_4.PART_A.STATUS.MASTER_PART := TRUE;
   END_IF;
   #_w8 := #_w1 AND "DB2099_MANUAL_LOAD_DMC".MANUAL_LOADING_OR_DRY_PART_UNLOADED_UNIT_02_P;
   #STATUS_FILL := FILL(EN := #_w8 AND NOT "DB2099_MANUAL_LOAD_DMC".PRODUCTION_SELECTED,
                        BVAL := #ZERO,
                        BLK => "DB8000_PART_STATUS".UNIT_02.FIXTURE_4.PART_A,
                        ENO => #_w9);
   IF #_w9 THEN
       "DB8000_PART_STATUS".UNIT_02.FIXTURE_4.PART_A.STATUS.PRESENT := FALSE;
       "DB8000_PART_STATUS".UNIT_02.FIXTURE_4.PART_A.STATUS.OK := FALSE;
   END_IF;
   #STATUS_BLKMOV := BLKMOV(EN := #_w8 AND "DB2099_MANUAL_LOAD_DMC".PRODUCTION_SELECTED,
                           SRCBLK := "DB8000_PART_STATUS".UNIT_02.FIXTURE_4.PART_A,
                           DSTBLK => "DB8101_MANUAL_LOADING_PART_STATUS_MANAGEMENT".UNIT_01_UNIT_02_INTERMEDIATE,
                           ENO => #_w10);
   #STATUS_FILL := FILL(EN := #_w10,
                        BVAL := #ZERO,
                        BLK => "DB8000_PART_STATUS".UNIT_02.FIXTURE_4.PART_A,
                        ENO => #_w11);
   IF #_w11 THEN
       "DB8101_MANUAL_LOADING_PART_STATUS_MANAGEMENT".UNIT_02_INTERMEDIATE.STATUS.PRESENT := TRUE;
       "DB8101_MANUAL_LOADING_PART_STATUS_MANAGEMENT".UNIT_02_INTERMEDIATE.STATUS.OK := TRUE;
       "DB8000_PART_STATUS".UNIT_02.FIXTURE_4.PART_A.STATUS.PRESENT := FALSE;
       "DB8000_PART_STATUS".UNIT_02.FIXTURE_4.PART_A.STATUS.OK := FALSE;
   END_IF;
END_REGION

REGION Network 24: INTERMEDIATE PARTS STATUS & PART ID RESET
   RUNG wire#powerrail
      I_Contact( "DB2099_MANUAL_LOAD_DMC".PRODUCTION_SELECTED )
      { S7_Templates := "ptr_type := Variant" } FILL(BVAL := #ZERO, RET_VAL => #STATUS_FILL, BLK => "DB8101_MANUAL_LOADING_PART_STATUS_MANAGEMENT".UNIT_01_INTERMEDIATE)
      { S7_Templates := "ptr_type := Variant" } FILL(BVAL := #ZERO, RET_VAL => #STATUS_FILL, BLK => "DB8101_MANUAL_LOADING_PART_STATUS_MANAGEMENT".UNIT_02_INTERMEDIATE)
      { S7_Templates := "ptr_type := Variant" } FILL(BVAL := #ZERO, RET_VAL => #STATUS_FILL, BLK => "DB8101_MANUAL_LOADING_PART_STATUS_MANAGEMENT".UNIT_01_UNIT_02_INTERMEDIATE)
   END_RUNG
   // the same network as SCL:
   #STATUS_FILL := FILL(EN := NOT "DB2099_MANUAL_LOAD_DMC".PRODUCTION_SELECTED,
                        BVAL := #ZERO,
                        BLK => "DB8101_MANUAL_LOADING_PART_STATUS_MANAGEMENT".UNIT_01_INTERMEDIATE,
                        ENO => #_w1);
   #STATUS_FILL := FILL(EN := #_w1,
                        BVAL := #ZERO,
                        BLK => "DB8101_MANUAL_LOADING_PART_STATUS_MANAGEMENT".UNIT_02_INTERMEDIATE,
                        ENO => #_w2);
   IF #_w2 THEN
       #STATUS_FILL := FILL(BVAL := #ZERO,
                            BLK => "DB8101_MANUAL_LOADING_PART_STATUS_MANAGEMENT".UNIT_01_UNIT_02_INTERMEDIATE);
   END_IF;
END_REGION
END_FUNCTION
